FUNCTION_BLOCK FB_SimulatedOutClose_DG IMPLEMENTS ITF_Regelschuif_OutClose_DG
VAR
	internalState : BOOL := FALSE;
END_VAR

{warning 'Add method implementation '}
METHOD set : BOOL
VAR_INPUT
	state : BOOL;
END_VAR
internalState := state;
END_METHOD

END_FUNCTION_BLOCK

(* stored: Version 1.1.0.1, ProductVersion 3.1.4026.8
   POU FB_SimulatedOutClose_DG: Id {097b5fdc-e3fa-4a76-920b-22891635337b}, SpecialFunc None
   Method set: Id {ab7d1b4f-9d6a-46ec-be20-89b919fc246a} *)
